(* IEC 61131-3 sources: FANUC_dev/LDJ/Kvara/PLC, 2 files *)

(* ---- Canfb.plc ---- *)
* Blocchi gestione periferiche CANopen da PLC

VAR_IN_OUT
AS_DATA0 AT %CanFb48; * CanFb48 buffer I/O Canopen
AS_DATA1 AT %CanFb49; * CanFb49 buffer I/O Canopen
AS_DATA2 AT %CanFb50; * CanFb50 buffer I/O Canopen
AS_DATA3 AT %CanFb51; * CanFb51 buffer I/O Canopen
AS_DATA4 AT %CanFb52; * CanFb52 buffer I/O Canopen
AS_DATA5 AT %CanFb53; * CanFb53 buffer I/O Canopen
AS_DATA6 AT %CanFb54; * CanFb54 buffer I/O Canopen
AS_DATA7 AT %CanFb55; * CanFb55 buffer I/O Canopen
DI_DATA0 AT %CanFb56; * CanFb56 Dato 0 input
DI_DATA1 AT %CanFb57; * CanFb57 Dato 1 input
DI_COBID AT %CanFb58; * CanFb58 Identificatore oggetto CanOpen
CONTROLREG AT %CanFb59; * CanFb59 registro comando (bit 0-7=codice comando)
CMD_RESET AT %CanFb59.30; * CanFb59.30 Reset nodo
CMD_ENAB AT %CanFb59.31; * CanFb59.31 Enable esecuzione comando
STATUSREG AT %CanFb60; * CanFb60 registro stato
DO_CONFIRM AT %CanFb60.31; * CanFb60.31 conferma comando eseguito
DO_ERROR AT %CanFb61; * CanFb61 codice errore comando
DO_DATA0 AT %CanFb62; * CanFb62 Dato 0 output
DO_DATA1 AT %CanFb63; * CanFb63 Dato 1 output
END_VAR

* -------------------------------------------------------*
* Blocco Funzionale generico invio comando a nodo CANopen
* -------------------------------------------------------*

FUNCTION_BLOCK COP_COMMAND

VAR_INPUT
CM_ENAB: BOOL; * Richiesta esecuzione comando
CM_RESET: BOOL; * Richiesta di reset del nodo
CM_CODE: DWORD; * Codice del comando
CI_COBID: DWORD; * Identificatore oggetto CanOpen
CI_DATA0: DWORD; * Dato 0 in input
CI_DATA1: DWORD; * Dato 1 in input
END_VAR

VAR_OUTPUT
CS_CONFIRM: BOOL; * Conferma comando eseguito
CO_ERROR: WORD; * Codice di errore
CO_ERRORINFO: DWORD; * Informazioni aggiuntive su errore
CO_DATA0: DWORD; * Dato 0 in output
CO_DATA1: DWORD; * Dato 1 in output
CO_DATA2: DWORD; * Dato 2 in output
CO_DATA3: DWORD; * Dato 3 in output
CO_DATA4: DWORD; * Dato 4 in output
CO_DATA5: DWORD; * Dato 5 in output
CO_DATA6: DWORD; * Dato 6 in output
CO_DATA7: DWORD; * Dato 7 in output
CO_DATA8: DWORD; * Dato 8 in output
END_VAR

VAR
StPrecEnab: BOOL; * Stato precedente ingresso ENAB
StPrecReset: BOOL; * Stato precedente ingresso RESET
StPrecConfirm: BOOL; * Stato precedente segnale CONFIRM
RTEnab: BOOL; * Fronte salita ingresso ENAB
MemCmdInProg: BOOL; * Mem. comando in corso
MemErrBusy: BOOL; * Mem. errore area comandi occupata
CmdFinished: BOOL; * Conferma comando terminato
END_VAR

* Sul fronte di salita del comando, copia tutti i dati in andata

LD   CM_ENAB      ** Richiesta esecuzione comando
ANDN StPrecEnab   ** Stato precedente ingresso ENAB
ST   RTEnab       ** Fronte salita ingresso ENAB

LD   RTEnab       ** Fronte salita ingresso ENAB
ANDN CMD_ENAB     ** CanFb59.31 Enable esecuzione comando
ANDN DO_CONFIRM   ** CanFb60.31 conferma comando eseguito
S    MemCmdInProg ** Mem. comando in corso

LDN  CM_ENAB      ** Richiesta esecuzione comando
ANDN CMD_ENAB     ** CanFb59.31 Enable esecuzione comando
ANDN DO_CONFIRM   ** CanFb60.31 conferma comando eseguito
OR   CM_RESET     ** Richiesta di reset del nodo
R    MemCmdInProg ** Mem. comando in corso

LD   RTEnab       ** Fronte salita ingresso ENAB
ANDN MemCmdInProg ** Mem. comando in corso
S    MemErrBusy   ** Mem. errore area comandi occupata

LDN  CM_ENAB      ** Richiesta esecuzione comando
R    MemErrBusy   ** Mem. errore area comandi occupata

LD   RTEnab       ** Fronte salita ingresso ENAB
AND  MemCmdInProg ** Mem. comando in corso
JMPCN END_COMMAND

LD   CONTROLREG   ** CanFb59 registro comando (bit 0-7=codice comando)
AND  16#FFFFFF00
OR   CM_CODE      ** Codice del comando
ST   CONTROLREG   ** CanFb59 registro comando (bit 0-7=codice comando)

LD   CI_COBID     ** Identificatore oggetto CanOpen
ST   DI_COBID     ** CanFb58 Identificatore oggetto CanOpen

LD   CM_CODE      ** Codice del comando
EQ   4            * PDO SEND
JMPC PDO_SEND_CMD

LD   CI_DATA0     ** Dato 0 in input
ST   DI_DATA0     ** CanFb56 Dato 0 input

LD   CI_DATA1     ** Dato 1 in input
ST   DI_DATA1     ** CanFb57 Dato 1 input

JMP  END_COMMAND

PDO_SEND_CMD:
LD   DI_COBID     ** CanFb58 Identificatore oggetto CanOpen
AND  16#FFFF00FF  * Mask offset
OR   16#3000      * Offset AS_DATA0 (48)
ST   DI_COBID     ** CanFb58 Identificatore oggetto CanOpen

LD   CI_DATA0     ** Dato 0 in input
ST   AS_DATA0     ** CanFb48 buffer I/O Canopen

LD   CI_DATA1     ** Dato 1 in input
ST   AS_DATA1     ** CanFb49 buffer I/O Canopen

END_COMMAND:

LD   CM_ENAB      ** Richiesta esecuzione comando
ST   StPrecEnab   ** Stato precedente ingresso ENAB

* Scrive i bit di ENAB e RESET

LD   MemCmdInProg ** Mem. comando in corso
JMPCN END_CMD_ENAB

LD   CM_ENAB      ** Richiesta esecuzione comando
ST   CMD_ENAB     ** CanFb59.31 Enable esecuzione comando

END_CMD_ENAB:

LD   CM_RESET     ** Richiesta di reset del nodo
OR   StPrecReset  ** Stato precedente ingresso RESET
JMPCN END_RESET

LD   CM_RESET     ** Richiesta di reset del nodo
ST   CMD_RESET    ** CanFb59.30 Reset nodo

LD   %PLCFLAGS.0
ST   CMD_ENAB     ** CanFb59.31 Enable esecuzione comando

END_RESET:

LD   CM_RESET     ** Richiesta di reset del nodo
ST   StPrecReset  ** Stato precedente ingresso RESET

* Sul fronte di salita della conferma fine comando, legge tutti i dati di ritorno

LD   DO_CONFIRM   ** CanFb60.31 conferma comando eseguito
AND  MemCmdInProg ** Mem. comando in corso
ST   CmdFinished  ** Conferma comando terminato

LD   DO_CONFIRM   ** CanFb60.31 conferma comando eseguito
ANDN StPrecConfirm ** Stato precedente segnale CONFIRM
AND  CmdFinished  ** Conferma comando terminato
JMPCN END_DATA

LD   DO_ERROR     ** CanFb61 codice errore comando
ST   CO_ERROR     ** Codice di errore

LD   DO_ERROR     ** CanFb61 codice errore comando
NE   0
JMPC TAKE_ERRINFO

LD   0
ST   CO_ERRORINFO ** Informazioni aggiuntive su errore

LD   CM_CODE      ** Codice del comando
EQ   5            * PDO READ
OR   (
LD   CM_CODE      ** Codice del comando
EQ   9            * SDO READSTR
)
OR   (
LD   CM_CODE      ** Codice del comando
EQ   10           * HISTORY ALARM
)
JMPC PDO_READ_CMD

LD   DO_DATA0     ** CanFb62 Dato 0 output
ST   CO_DATA0     ** Dato 0 in output

LD   DO_DATA1     ** CanFb63 Dato 1 output
ST   CO_DATA1     ** Dato 1 in output

JMP  END_DATA

PDO_READ_CMD:

LD   DO_DATA0     ** CanFb62 Dato 0 output
ST   CO_DATA0     ** Dato 0 in output

LD   AS_DATA0     ** CanFb48 buffer I/O Canopen
ST   CO_DATA1     ** Dato 1 in output

LD   AS_DATA1     ** CanFb49 buffer I/O Canopen
ST   CO_DATA2     ** Dato 2 in output

LD   CM_CODE      ** Codice del comando
EQ   5            * PDO READ
JMPC END_DATA

LD   AS_DATA2     ** CanFb50 buffer I/O Canopen
ST   CO_DATA3     ** Dato 3 in output

LD   AS_DATA3     ** CanFb51 buffer I/O Canopen
ST   CO_DATA4     ** Dato 4 in output

LD   AS_DATA4     ** CanFb52 buffer I/O Canopen
ST   CO_DATA5     ** Dato 5 in output

LD   AS_DATA5     ** CanFb53 buffer I/O Canopen
ST   CO_DATA6     ** Dato 6 in output

LD   AS_DATA6     ** CanFb54 buffer I/O Canopen
ST   CO_DATA7     ** Dato 7 in output

LD   AS_DATA7     ** CanFb55 buffer I/O Canopen
ST   CO_DATA8     ** Dato 8 in output

JMP  END_DATA

TAKE_ERRINFO:

LD   DO_DATA0     ** CanFb62 Dato 0 output
ST   CO_ERRORINFO ** Informazioni aggiuntive su errore

LD   0
ST   CO_DATA0     ** Dato 0 in output
ST   CO_DATA1     ** Dato 1 in output

END_DATA:

LD   MemErrBusy   ** Mem. errore area comandi occupata
JMPCN END_TR_ERR

LD   16#25        * Errore TRANSFER_BUSY
ST   CO_ERROR     ** Codice di errore

END_TR_ERR:

* Scrive in output la conferma

LD   DO_CONFIRM   ** CanFb60.31 conferma comando eseguito
ST   StPrecConfirm ** Stato precedente segnale CONFIRM

LD   CmdFinished  ** Conferma comando terminato
OR   MemErrBusy   ** Mem. errore area comandi occupata
ST   CS_CONFIRM   ** Conferma comando eseguito

END_FUNCTION_BLOCK

* -------------------------------------------------------*
* Comando di cambio di stato a nodo CANopen
* -------------------------------------------------------*

FUNCTION_BLOCK COP_NMT

VAR_INPUT
CM_ENAB: BOOL; * Richiesta esecuzione comando
CM_RESET: BOOL; * Richiesta di reset del nodo
CI_STATE: DWORD; * Stato richiesto
END_VAR

VAR_OUTPUT
CS_CONFIRM: BOOL; * Conferma comando eseguito
CO_ERROR: WORD; * Codice di errore
END_VAR

VAR
COPFB: COP_COMMAND;
END_VAR

LD   CM_ENAB      ** Richiesta esecuzione comando
ST   COPFB.CM_ENAB

LD   CM_RESET     ** Richiesta di reset del nodo
ST   COPFB.CM_RESET

LD   1
ST   COPFB.CM_CODE

LD   CI_STATE     ** Stato richiesto
ST   COPFB.CI_DATA0

CAL  COPFB

LD   COPFB.CS_CONFIRM
ST   CS_CONFIRM   ** Conferma comando eseguito

LD   COPFB.CO_ERROR
ST   CO_ERROR     ** Codice di errore

END_FUNCTION_BLOCK

* -------------------------------------------------------*
* Comando di lettura SDO a nodo CANopen
* -------------------------------------------------------*

FUNCTION_BLOCK COP_SDO_READ

VAR_INPUT
CM_ENAB: BOOL; * Richiesta esecuzione comando
CM_RESET: BOOL; * Richiesta di reset del nodo
CI_INDEX: DWORD; * Numero index dato da leggere
CI_SUBINDEX: DWORD; * Numero subindex dato da leggere
END_VAR

VAR_OUTPUT
CS_CONFIRM: BOOL; * Conferma comando eseguito
CO_ERROR: WORD; * Codice di errore
CO_ERRORINFO: DWORD; * Informazioni aggiuntive su errore
CO_DATALENGTH: DWORD; * Lunghezza dato letto in byte
CO_DATA0: DWORD; * Valore del dato letto
END_VAR

VAR
COPFB: COP_COMMAND;
END_VAR

LD   CM_ENAB      ** Richiesta esecuzione comando
ST   COPFB.CM_ENAB

LD   CM_RESET     ** Richiesta di reset del nodo
ST   COPFB.CM_RESET

LD   2
ST   COPFB.CM_CODE

LD   CI_INDEX     ** Numero index dato da leggere
SHL  16
OR   (
LD   CI_SUBINDEX  ** Numero subindex dato da leggere
SHL  8
)
ST   COPFB.CI_COBID

CAL  COPFB

LD   COPFB.CS_CONFIRM
ST   CS_CONFIRM   ** Conferma comando eseguito

LD   COPFB.CO_ERROR
ST   CO_ERROR     ** Codice di errore

LD   COPFB.CO_ERRORINFO
ST   CO_ERRORINFO ** Informazioni aggiuntive su errore

LD   COPFB.CO_DATA0
ST   CO_DATALENGTH ** Lunghezza dato letto in byte

LD   COPFB.CO_DATA1
ST   CO_DATA0     ** Valore del dato letto

END_FUNCTION_BLOCK

* -------------------------------------------------------*
* Comando di scrittura SDO a nodo CANopen
* -------------------------------------------------------*

FUNCTION_BLOCK COP_SDO_WRITE

VAR_INPUT
CM_ENAB: BOOL; * Richiesta esecuzione comando
CM_RESET: BOOL; * Richiesta di reset del nodo
CI_INDEX: DWORD; * Numero index dato da scrivere
CI_SUBINDEX: DWORD; * Numero subindex dato da scrivere
CI_DATALENGTH: DWORD; * Lunghezza dato da scrivere in byte
CI_DATA0: DWORD; * Valore da scrivere
END_VAR

VAR_OUTPUT
CS_CONFIRM: BOOL; * Conferma comando eseguito
CO_ERROR: WORD; * Codice di errore
CO_ERRORINFO: DWORD; * Informazioni aggiuntive su errore
END_VAR

VAR
COPFB: COP_COMMAND;
END_VAR

LD   CM_ENAB      ** Richiesta esecuzione comando
ST   COPFB.CM_ENAB

LD   CM_RESET     ** Richiesta di reset del nodo
ST   COPFB.CM_RESET

LD   3
ST   COPFB.CM_CODE

LD   CI_INDEX     ** Numero index dato da scrivere
SHL  16
OR   (
LD   CI_SUBINDEX  ** Numero subindex dato da scrivere
SHL  8
)
OR   CI_DATALENGTH ** Lunghezza dato da scrivere in byte
ST   COPFB.CI_COBID

LD   CI_DATA0     ** Valore da scrivere
ST   COPFB.CI_DATA0

CAL  COPFB

LD   COPFB.CS_CONFIRM
ST   CS_CONFIRM   ** Conferma comando eseguito

LD   COPFB.CO_ERROR
ST   CO_ERROR     ** Codice di errore

LD   COPFB.CO_ERRORINFO
ST   CO_ERRORINFO ** Informazioni aggiuntive su errore

END_FUNCTION_BLOCK

* -------------------------------------------------------*
* Comando di invio PDO a nodo CANopen
* -------------------------------------------------------*

FUNCTION_BLOCK COP_PDO_SEND

VAR_INPUT
CM_ENAB: BOOL; * Richiesta esecuzione comando
CM_RESET: BOOL; * Richiesta di reset del nodo
CI_COBID: DWORD; * Identificatore oggetto CanOpen
CI_DATALENGTH: DWORD; * Lunghezza dato da scrivere in byte
CI_DATA0: DWORD; * Valore da inviare (BYTE 0-3)
CI_DATA1: DWORD; * Valore da inviare (BYTE 4-7)
END_VAR

VAR_OUTPUT
CS_CONFIRM: BOOL; * Conferma comando eseguito
CO_ERROR: WORD; * Codice di errore
END_VAR

VAR
COPFB: COP_COMMAND;
END_VAR

LD   CM_ENAB      ** Richiesta esecuzione comando
ST   COPFB.CM_ENAB

LD   CM_RESET     ** Richiesta di reset del nodo
ST   COPFB.CM_RESET

LD   4
ST   COPFB.CM_CODE

LD   CI_COBID     ** Identificatore oggetto CanOpen
SHL  16
OR   CI_DATALENGTH ** Lunghezza dato da scrivere in byte
ST   COPFB.CI_COBID

LD   CI_DATA0     ** Valore da inviare (BYTE 0-3)
ST   COPFB.CI_DATA0

LD   CI_DATA1     ** Valore da inviare (BYTE 4-7)
ST   COPFB.CI_DATA1

CAL  COPFB

LD   COPFB.CS_CONFIRM
ST   CS_CONFIRM   ** Conferma comando eseguito

LD   COPFB.CO_ERROR
ST   CO_ERROR     ** Codice di errore

END_FUNCTION_BLOCK

* -------------------------------------------------------*
* Comando di lettura PDO da nodo CANopen
* -------------------------------------------------------*

FUNCTION_BLOCK COP_PDO_READ

VAR_INPUT
CM_ENAB: BOOL; * Richiesta esecuzione comando
CM_RESET: BOOL; * Richiesta di reset del nodo
CI_COBID: DWORD; * Identificatore oggetto CanOpen
END_VAR

VAR_OUTPUT
CS_CONFIRM: BOOL; * Conferma comando eseguito
CO_ERROR: WORD; * Codice di errore
CO_DATALENGTH: DWORD; * Lunghezza PDO letto in byte
CO_DATA0: DWORD; * Valore del dato letto (BYTE 0-3)
CO_DATA1: DWORD; * Valore del dato letto (BYTE 4-7)
END_VAR

VAR
COPFB: COP_COMMAND;
END_VAR

LD   CM_ENAB      ** Richiesta esecuzione comando
ST   COPFB.CM_ENAB

LD   CM_RESET     ** Richiesta di reset del nodo
ST   COPFB.CM_RESET

LD   5
ST   COPFB.CM_CODE

LD   CI_COBID     ** Identificatore oggetto CanOpen
SHL  16
ST   COPFB.CI_COBID

CAL  COPFB

LD   COPFB.CS_CONFIRM
ST   CS_CONFIRM   ** Conferma comando eseguito

LD   COPFB.CO_ERROR
ST   CO_ERROR     ** Codice di errore

LD   COPFB.CO_DATA0
ST   CO_DATALENGTH ** Lunghezza PDO letto in byte

LD   COPFB.CO_DATA1
ST   CO_DATA0     ** Valore del dato letto (BYTE 0-3)

LD   COPFB.CO_DATA2
ST   CO_DATA1     ** Valore del dato letto (BYTE 4-7)

END_FUNCTION_BLOCK

* -------------------------------------------------------*
* Comando di registrazione PDO
* -------------------------------------------------------*

FUNCTION_BLOCK COP_PDO_REGISTER

VAR_INPUT
CM_ENAB: BOOL; * Richiesta esecuzione comando
CM_RESET: BOOL; * Richiesta di reset del nodo
CI_COBID: DWORD; * Identificatore oggetto CanOpen
CI_DATALENGTH: DWORD; * Lunghezza in BYTE e tipo dato (FFFF = cancella registr.)
                      * lungh + 0: legge con COP_PDO_READ
                      * lungh + 256: legge da CanFb0-CanFb47
                      * lungh + 512: legge da IW0-IW2047
CI_DATAOFFSET: DWORD; * Offset rinfresco (CanFb[0-47] / IO[0-2047])
END_VAR

VAR_OUTPUT
CS_CONFIRM: BOOL; * Conferma comando eseguito
CO_ERROR: WORD; * Codice di errore
END_VAR

VAR
COPFB: COP_COMMAND;
END_VAR

LD   CM_ENAB      ** Richiesta esecuzione comando
ST   COPFB.CM_ENAB

LD   CM_RESET     ** Richiesta di reset del nodo
ST   COPFB.CM_RESET

LD   6
ST   COPFB.CM_CODE

LD   CI_COBID     ** Identificatore oggetto CanOpen
SHL  16
OR   CI_DATALENGTH ** Lunghezza in BYTE e tipo dato (FFFF = cancella registr.)
ST   COPFB.CI_COBID

LD   CI_DATAOFFSET ** Offset rinfresco (CanFb[0-47] / IO[0-2047])
ST   COPFB.CI_DATA0

CAL  COPFB

LD   COPFB.CS_CONFIRM
ST   CS_CONFIRM   ** Conferma comando eseguito

LD   COPFB.CO_ERROR
ST   CO_ERROR     ** Codice di errore

END_FUNCTION_BLOCK

* -------------------------------------------------------*
* Comando di impostazione sincronizzazione ciclica
* -------------------------------------------------------*

FUNCTION_BLOCK COP_CYCLIC_SYNC

VAR_INPUT
CM_ENAB: BOOL; * Richiesta esecuzione comando
CM_RESET: BOOL; * Richiesta di reset del nodo
CI_SYNC_TIME: DWORD; * Tempo ciclo (0=Disab, 1=Singolo, 10-250=Ciclico in ms)
END_VAR

VAR_OUTPUT
CS_CONFIRM: BOOL; * Conferma comando eseguito
CO_ERROR: WORD; * Codice di errore
END_VAR

VAR
COPFB: COP_COMMAND;
END_VAR

LD   CM_ENAB      ** Richiesta esecuzione comando
ST   COPFB.CM_ENAB

LD   CM_RESET     ** Richiesta di reset del nodo
ST   COPFB.CM_RESET

LD   7
ST   COPFB.CM_CODE

LD   CI_SYNC_TIME ** Tempo ciclo (0=Disab, 1=Singolo, 10-250=Ciclico in ms)
ST   COPFB.CI_DATA0

CAL  COPFB

LD   COPFB.CS_CONFIRM
ST   CS_CONFIRM   ** Conferma comando eseguito

LD   COPFB.CO_ERROR
ST   CO_ERROR     ** Codice di errore

END_FUNCTION_BLOCK

* -------------------------------------------------------*
* Comando di remote request oggetto CANopen
* -------------------------------------------------------*

FUNCTION_BLOCK COP_REM_REQUEST

VAR_INPUT
CM_ENAB: BOOL; * Richiesta esecuzione comando
CM_RESET: BOOL; * Richiesta di reset del nodo
CI_COBID: DWORD; * Identificatore oggetto CanOpen
END_VAR

VAR_OUTPUT
CS_CONFIRM: BOOL; * Conferma comando eseguito
CO_ERROR: WORD; * Codice di errore
END_VAR

VAR
COPFB: COP_COMMAND;
END_VAR

LD   CM_ENAB      ** Richiesta esecuzione comando
ST   COPFB.CM_ENAB

LD   CM_RESET     ** Richiesta di reset del nodo
ST   COPFB.CM_RESET

LD   8
ST   COPFB.CM_CODE

LD   CI_COBID     ** Identificatore oggetto CanOpen
ST   COPFB.CI_COBID

CAL  COPFB

LD   COPFB.CS_CONFIRM
ST   CS_CONFIRM   ** Conferma comando eseguito

LD   COPFB.CO_ERROR
ST   CO_ERROR     ** Codice di errore

END_FUNCTION_BLOCK

* -------------------------------------------------------*
* Comando di lettura SDO su stringa da nodo CANopen
* -------------------------------------------------------*

FUNCTION_BLOCK COP_SDO_READSTRING

VAR_INPUT
CM_ENAB: BOOL; * Richiesta esecuzione comando
CM_RESET: BOOL; * Richiesta di reset del nodo
CI_INDEX: DWORD; * Numero index dato da leggere
CI_SUBINDEX: DWORD; * Numero subindex dato da leggere
END_VAR

VAR_OUTPUT
CS_CONFIRM: BOOL; * Conferma comando eseguito
CO_ERROR: WORD; * Codice di errore
CO_ERRORINFO: DWORD; * Informazioni aggiuntive su errore
CO_DATALENGTH: DWORD; * Lunghezza stringa letta in byte
CO_DATA0: DWORD; * Stringa letta (BYTE 0-3)
CO_DATA1: DWORD; * Stringa letta (BYTE 4-7)
CO_DATA2: DWORD; * Stringa letta (BYTE 8-11)
CO_DATA3: DWORD; * Stringa letta (BYTE 12-15)
CO_DATA4: DWORD; * Stringa letta (BYTE 16-19)
CO_DATA5: DWORD; * Stringa letta (BYTE 20-23)
CO_DATA6: DWORD; * Stringa letta (BYTE 24-27)
CO_DATA7: DWORD; * Stringa letta (BYTE 28-31)
END_VAR

VAR
COPFB: COP_COMMAND;
END_VAR

LD   CM_ENAB      ** Richiesta esecuzione comando
ST   COPFB.CM_ENAB

LD   CM_RESET     ** Richiesta di reset del nodo
ST   COPFB.CM_RESET

LD   9
ST   COPFB.CM_CODE

LD   CI_INDEX     ** Numero index dato da leggere
SHL  16
OR   (
LD   CI_SUBINDEX  ** Numero subindex dato da leggere
SHL  8
)
ST   COPFB.CI_COBID

CAL  COPFB

LD   COPFB.CS_CONFIRM
ST   CS_CONFIRM   ** Conferma comando eseguito

LD   COPFB.CO_ERROR
ST   CO_ERROR     ** Codice di errore

LD   COPFB.CO_ERRORINFO
ST   CO_ERRORINFO ** Informazioni aggiuntive su errore

LD   COPFB.CO_DATA0
ST   CO_DATALENGTH ** Lunghezza stringa letta in byte

LD   COPFB.CO_DATA1
ST   CO_DATA0     ** Stringa letta (BYTE 0-3)

LD   COPFB.CO_DATA2
ST   CO_DATA1     ** Stringa letta (BYTE 4-7)

LD   COPFB.CO_DATA3
ST   CO_DATA2     ** Stringa letta (BYTE 8-11)

LD   COPFB.CO_DATA4
ST   CO_DATA3     ** Stringa letta (BYTE 12-15)

LD   COPFB.CO_DATA5
ST   CO_DATA4     ** Stringa letta (BYTE 16-19)

LD   COPFB.CO_DATA6
ST   CO_DATA5     ** Stringa letta (BYTE 20-23)

LD   COPFB.CO_DATA7
ST   CO_DATA6     ** Stringa letta (BYTE 24-27)

LD   COPFB.CO_DATA8
ST   CO_DATA7     ** Stringa letta (BYTE 28-31)

END_FUNCTION_BLOCK

* -------------------------------------------------------*
* Comando Read/Reset History alarm da nodo CANopen
* -------------------------------------------------------*

FUNCTION_BLOCK COP_ALARMS_HIST

VAR_INPUT
CM_ENAB:  BOOL; * Richiesta esecuzione comando
CM_RESET: BOOL; * Richiesta di reset del nodo
CI_MODE:  BOOL; * 0=Read  1=Read & Reset
END_VAR

VAR_OUTPUT
CS_CONFIRM: BOOL; * Conferma comando eseguito
CO_ERROR:   WORD; * Codice di errore
CO_ERRORINFO: DWORD;  * Informazioni aggiuntive su errore
CO_ALARMS:    DWORD;  * Numero di allarmi presenti
CO_ALRM1: DWORD; * Ultimo allarme "n"
CO_ALRM2: DWORD; * Allarme "n-1"
CO_ALRM3: DWORD; * Allarme "n-2"
CO_ALRM4: DWORD; * Allarme "n-3"
CO_ALRM5: DWORD; * Allarme "n-4"
CO_ALRM6: DWORD; * Allarme "n-5"
CO_ALRM7: DWORD; * Allarme "n-6"
CO_ALRM8: DWORD; * Allarme "n-7"
END_VAR

VAR
COPFB: COP_COMMAND;
END_VAR

LD   CM_ENAB      ** Richiesta esecuzione comando
ST   COPFB.CM_ENAB

LD   CM_RESET     ** Richiesta di reset del nodo
ST   COPFB.CM_RESET

LD   10
ST   COPFB.CM_CODE

LD   CI_MODE      ** 0=Read  1=Read & Reset
ST   COPFB.CI_DATA0.0   ** CanFb56 Dato 0 input

CAL  COPFB

LD   COPFB.CS_CONFIRM
ST   CS_CONFIRM   ** Conferma comando eseguito

LD   COPFB.CO_ERROR
ST   CO_ERROR     ** Codice di errore

LD   COPFB.CO_ERRORINFO
ST   CO_ERRORINFO ** Informazioni aggiuntive su errore

LD   DO_DATA0     ** CanFb62 Dato 0 output
ST   CO_ALARMS    ** Numero di allarmi presenti

LD   COPFB.CO_DATA1
ST   CO_ALRM1     ** Ultimo allarme "n"

LD   COPFB.CO_DATA2
ST   CO_ALRM2     ** Allarme "n-1"

LD   COPFB.CO_DATA3
ST   CO_ALRM3     ** Allarme "n-2"

LD   COPFB.CO_DATA4
ST   CO_ALRM4     ** Allarme "n-3"

LD   COPFB.CO_DATA5
ST   CO_ALRM5     ** Allarme "n-4"

LD   COPFB.CO_DATA6
ST   CO_ALRM6     ** Allarme "n-5"

LD   COPFB.CO_DATA7
ST   CO_ALRM7     ** Allarme "n-6"

LD   COPFB.CO_DATA8
ST   CO_ALRM8     ** Allarme "n-7"

END_FUNCTION_BLOCK

* -------------------------------------------------------*
* Comando di lettura VACON ReadAnyParam
* -------------------------------------------------------*

FUNCTION_BLOCK VAC_PAR_READ

VAR_INPUT
CM_ENAB: BOOL; * Richiesta esecuzione comando
CM_RESET: BOOL; * Richiesta di reset del nodo
CI_INDEX: DWORD; * Numero parametro da leggere
END_VAR

VAR_OUTPUT
CS_CONFIRM: BOOL; * Conferma comando eseguito
CO_ERROR: WORD; * Codice di errore
CO_ERRORINFO: DWORD; * Informazioni aggiuntive su errore
CO_DATALENGTH: DWORD; * Lunghezza dato letto in byte
CO_DATA0: DWORD; * Valore del dato letto
END_VAR

VAR
COPFB: COP_COMMAND;
END_VAR

LD   CM_ENAB      ** Richiesta esecuzione comando
ST   COPFB.CM_ENAB

LD   CM_RESET     ** Richiesta di reset del nodo
ST   COPFB.CM_RESET

LD   255
ST   COPFB.CM_CODE

LD   CI_INDEX     ** Numero index dato da leggere
ST   COPFB.CI_COBID

CAL  COPFB

LD   COPFB.CS_CONFIRM
ST   CS_CONFIRM   ** Conferma comando eseguito

LD   COPFB.CO_ERROR
ST   CO_ERROR     ** Codice di errore

LD   COPFB.CO_ERRORINFO
ST   CO_ERRORINFO ** Informazioni aggiuntive su errore

LD   COPFB.CO_DATA0
ST   CO_DATALENGTH ** Lunghezza dato letto in byte

LD   COPFB.CO_DATA1
ST   CO_DATA0     ** Valore del dato letto

END_FUNCTION_BLOCK

* -------------------------------------------------------*
* Comando di scrittura VACON WriteAnyParam
* -------------------------------------------------------*

FUNCTION_BLOCK VAC_PAR_WRITE

VAR_INPUT
CM_ENAB: BOOL; * Richiesta esecuzione comando
CM_RESET: BOOL; * Richiesta di reset del nodo
CI_INDEX: DWORD; * Numero parametro dato da scrivere
CI_DATA0: DWORD; * Valore da scrivere
END_VAR

VAR_OUTPUT
CS_CONFIRM: BOOL; * Conferma comando eseguito
CO_ERROR: WORD; * Codice di errore
CO_ERRORINFO: DWORD; * Informazioni aggiuntive su errore
END_VAR

VAR
COPFB: COP_COMMAND;
END_VAR

LD   CM_ENAB      ** Richiesta esecuzione comando
ST   COPFB.CM_ENAB

LD   CM_RESET     ** Richiesta di reset del nodo
ST   COPFB.CM_RESET

LD   254
ST   COPFB.CM_CODE

LD   CI_INDEX     ** Numero index dato da scrivere
ST   COPFB.CI_COBID

LD   CI_DATA0     ** Valore da scrivere
ST   COPFB.CI_DATA0

CAL  COPFB

LD   COPFB.CS_CONFIRM
ST   CS_CONFIRM   ** Conferma comando eseguito

LD   COPFB.CO_ERROR
ST   CO_ERROR     ** Codice di errore

LD   COPFB.CO_ERRORINFO
ST   CO_ERRORINFO ** Informazioni aggiuntive su errore

END_FUNCTION_BLOCK

(* ---- usercmd.plc ---- *)
* File USERCMD.PLC

#include "iof.inc"
#include "iol.inc"
#include "mem.inc"

VAR
IN_LUBR_ERR    AT %IW0.13;  * IW0.13 Errore Centralina Lubrificazione (cartuccia Vuota)
LUBR_ERR: BOOL;              * IW0.13 Errore Centralina Lubrificazione (cartuccia Vuota) Solo quando lubrificazzione in corso
LUBR_OK     AT %IW0.14;  * IW0.14 Lubrificazione OK
IN_CELLA_APERTA AT %IW3.8; * IW3.8 Ingresso Cella Aperta
BRAKE_OPEN  AT %IW3.0;   * IW3.0 Freni aperti, consenso al movimento Ok
STOP_PCV    AT %IW3.3;   * IW3.3 Blocco ciclo al PCV
STOP_PCL    AT %IW3.4;   * IW3.4 Blocco ciclo al PCL dopo il rinculo
STOP_PMI    AT %IW3.5;   * IW3.5 Blocco ciclo al PMI dopo il tempo sosta
LUBR_REQ    AT %QW1.8;   * QW1.8 Richiesta Lubrificazione
FIRST_BEND  AT %QW2.13;  * QW2.13 Prima Piega Attiva
PMS_ROBOT   AT %QW2.8;   * QW2.8 PMS per Robot
OUT_INT_LAMP AT %QW1.10; * QW1.10 Uscita Accensione Lampada Interna
PUMP_ON_PUNCH_HOLDER AT %QW1.11; * Uscita Attivazione Pompa Bloccaggi Superiori
PUMP_ON_DIE_HOLDER   AT %QW1.12; * Uscita Attivazione Pompa Bloccaggi Inferiori o Bloccaggio Singolo
HOLDER_OPENED        AT %QW1.13; * Uscita Bloccaggi Aperti
PUNCH_HOLDER_OPENED  AT %QW1.14; * Uscita Bloccaggi Superiori Aperti
DIE_HOLDER_OPENED    AT %QW1.15; * Uscita Bloccaggi Inferiori Aperti
ANIN2       AT %IW51;    * Ingresso analogico Pin 2
ANIN3       AT %IW52;    * Ingresso analogico Pin 3
VOLT_LED    AT %QW102;   * QW102 Tensione regolazione intensità luminosa Lampada

Cond_Cont_Lubr: BOOL; * Condizione Conteggio Lubrificazione
Cond_Reload_Cont: BOOL; * Condizione Reload Conteggio Lubrificazione
Param_Changed: BOOL; * Parametro Cambiato
LUB_ERR_REMIND: BOOL; * Reminder Cartuccia Lubrificazione Terminata
LubrErr: BOOL; * Cartuccia Vuota
Lubrinproc: BOOL; * Cartuccia Vuota stato in memoria
VLED_0_BIT: WORD; * Tensione Lampada 0% in Bit
VLED_100_BIT: WORD; * Tensione Lampada 100% in Bit

***** Limitazione Sbilanciamento in Discesa Lenta *****
Y1_STOP_UNBALANCE: BOOL; * Necessario Stop Y1 per sbilanciamento eccessivo
Y2_STOP_UNBALANCE: BOOL; * Necessario Stop Y2 per sbilanciamento eccessivo
Y1_FEED_CALC: WORD; * Valore Feed Y1 Ricalcolata
Y2_FEED_CALC: WORD; * Valore Feed Y2 Ricalcolata
***** Fine Limitazione Sbilanciamento in Discesa Lenta *****

TON_FILTER: TON;
#defcom TON_FILTER.Q Filtro per pedale di discesa
#defcom CTD_LUBR.Q Fine Conteggio per attivazione lubrificazione
#defcom CTD_LUBR.CV Stato del Contatore Lubrificazione
CTD_LUBR: CTD;
#defcom CTD_LUBR_OK.Q Fine Conteggio per check lubrificazione
CTD_LUBR_OK: CTD;
#defcom TP_LUBR.Q    Tempo Uscita Lubrificazione Attiva
TP_LUBR: TP;
#defcom TOF_LUBR_EMPTY.Q    Cartuccia Vuota
TOF_LUBR_EMPTY: TOF;
#defcom R_TRIG_LUBR.Q Fronte salita Richiesta Lubrificazione
R_TRIG_LUBR: R_TRIG;
#defcom TRIG_LUBR_OK.Q Fronte salita Ingresso Lubrificazione in corso
TRIG_LUBR_OK: TRIG;
#defcom F_TRIG_LUBREMPTY.Q Fronte discesa Cartuccia vuota
F_TRIG_LUBREMPTY: F_TRIG;

#defcom TOF_PRES_SUP.Q    Filtro apertura bloccaggi superiori
TOF_PRES_SUP: TOF;
#defcom TOF_PRES_INF.Q    Filtro apertura bloccaggi inferiori
TOF_PRES_INF: TOF;

#defcom %paruser.dwuser0     Numero cicli per lubrificazione
#defcom %paruser.dwuser1     Tensione Lampada allo 0%
#defcom %paruser.dwuser2     Tensione Lampada al 100%
#defcom %paruser.buser.0     Bloccaggi Singolo
#defcom %paruser.buser.1     Bloccaggi Doppio
V_MAX_CLOSE_TOOLS AT %paruser.dwuser4;   * Tensione Massima per Attivazione Pompa
V_MIN_CLOSE_TOOLS AT %paruser.dwuser5;   * Tensione Minima per Attivazione Pompa
V_TOOLS_OPENED    AT %paruser.dwuser6;   * Tensione Utensili Aperti

#defcom %PLCerr3.3    Allarme Richiesta Lubrificazione, Centralina non risponde
#defcom %PLCerr3.4    Allarme Cartuccia Danneggiata
#defcom %PLCerr3.5    Allarme Cartuccia Vuota
#defcom %PLCerr3.6    Allarme Freni Chiusi

END_VAR

VAR_IN_OUT

INTERNAL_LIGTH  AT %R65.0;   * R65.0 Pulsante UI accensione / spegnimento Lampada interna
VOUT_LED        AT %R64;     * R64 Tensione Bit in uscita
COUNT_LUBR_MEM  AT %R63;     * R63 Parametro Conteggio Lubrificazione in Memoria
Lubrinprocmem   AT %R62.0;   * Cartuccia vuota stato in memoria
COUNT_LUBR_CV   AT %M127;    * M127 Strokes Left for Lubrification
PERC_V_LED      AT %M128;    * M128 Percentuale Tensione LED
VOLT_LED_DEC    AT %M129.0;  * M129.0 Pulsante decremento Tensione LED 1%
VOLT_LED_INC    AT %M129.1;  * M129.1 Pulsante incremento Tensione LED 1%
VOLT_LED_DEC10  AT %M129.2;  * M129.2 Pulsante decremento Tensione LED 10%
VOLT_LED_INC10  AT %M129.3;  * M129.3 Pulsante incremento Tensione LED 10%
VOLT_LED_OFF    AT %M129.4;  * M129.4 Pulsante spegnimento Lamada
VOLT_LED_100    AT %M129.5;  * M129.5 Pulsante accensione Lampada al 100%
COUNTER         AT %paruser.dwuser0; ** Numero cicli per lubrificazione

END_VAR

* Funzione utente per la gestione di input ausiliari e il forzamento
* di input per il programma MAIN.

FUNCTION USERIN

** Filtro per pedale discesa Starmatik **

*CAL   TON_FILTER(IN=%C60.0, PT=300)

*LD    TON_FILTER.Q
*ST    %C60.0

*CAL   TOF_PRES_SUP(IN=%C61.26, PT=1000)  * IN Pressostato bloccaggi superiori
*CAL   TOF_PRES_INF(IN=%C61.27, PT=1000)  * IN Pressostato bloccaggi inferiori

*LD    TOF_PRES_SUP.Q
*ST    %C61.26   * IN Pressostato bloccaggi superiori

*LD    TOF_PRES_INF.Q
*ST    %C61.27   * IN Pressostato bloccaggi inferiori

LDN    %C62.20   ** Allarme Utente 2
ST     %C62.20   ** Allarme Utente 2

END_FUNCTION

* Funzione utente per il comando di segnalazioni e uscite ausiliarie.

FUNCTION USERCMD

* Esempio
*LD   %IW0.0
*ST   %PLCerr3.0

************************** Gestione Lubrificazione ***********************************

LD   IN_LUBR_ERR     * IW0.13 Errore Centralina Lubrificazione (cartuccia Vuota)
ORN  LUBR_REQ        ** QW1.8 Richiesta Lubrificazione
ST   LUBR_ERR        * IW0.13 Errore Centralina Lubrificazione (cartuccia Vuota) Solo quando lubrificazzione in corso

LD   %paruser.dwuser0 ** Numero cicli per lubrificazione
EQ   0
JMPC NOLUBR

LD   %C70.16      ** OUT Macchina al PMS
ST   Cond_Cont_Lubr ** Condizione Conteggio Lubrificazione

LD   COUNTER      ** Parametro Conteggio Lubrificazione
EQ   COUNT_LUBR_MEM ** R63 Parametro Conteggio Lubrificazione in Memoria
JMPC PARAM_NOT_CHANGED

LD   %PLCFLAGS.1  ** Sempre a uno
ST   Param_Changed ** Parametro Cambiato

LD   COUNTER      ** Parametro Conteggio Lubrificazione
ST   COUNT_LUBR_MEM ** R63 Parametro Conteggio Lubrificazione in Memoria

PARAM_NOT_CHANGED:

LD   CTD_LUBR.Q   ** Fine Conteggio per attivazione lubrificazione
OR   Param_Changed ** Parametro Cambiato
ST   Cond_Reload_Cont ** Condizione Reload Conteggio Lubrificazione

LD   %PLCFLAGS.0  ** Sempre a zero
ST   Param_Changed ** Parametro Cambiato

CAL  CTD_LUBR(CD:=Cond_Cont_Lubr, LD:=Cond_Reload_Cont , PV:=%paruser.dwuser0) ** Condizione Conteggio Lubrificazione

CAL  TP_LUBR(IN=CTD_LUBR.Q,PT=10000) ** Fine Conteggio per attivazione lubrificazione

CAL  R_TRIG_LUBR(CLK=TP_LUBR.Q) ** Tempo Uscita Lubrificazione Attiva

CAL  F_TRIG_LUBREMPTY(CLK=LUBR_ERR) ** IW0.13 Errore Centralina Lubrificazione (cartuccia Vuota)

CAL  TRIG_LUBR_OK(CLK=LUBR_OK) ** IW0.14 Lubrificazione OK

CAL  CTD_LUBR_OK(CD:=TRIG_LUBR_OK.Q, LD:=R_TRIG_LUBR.Q , PV:=1) ** Fronte salita Ingresso Lubrificazione in corso

LD   R_TRIG_LUBR.Q ** Fronte salita Richiesta Lubrificazione
S    Lubrinprocmem ** Cartuccia vuota stato in memoria

LD   R_TRIG_LUBR.Q ** Fronte salita Richiesta Lubrificazione
OR   (
LD   Lubrinprocmem ** Cartuccia vuota stato in memoria
AND  %PLCFLAGS.8  ** Bit a uno alla prima scansione
)
S    Lubrinproc   ** Cartuccia Vuota stato in memoria

LD   CTD_LUBR_OK.Q ** Fine Conteggio per check lubrificazione
R    Lubrinprocmem ** Cartuccia vuota stato in memoria

LD   CTD_LUBR_OK.Q ** Fine Conteggio per check lubrificazione
OR   %M5.5         ** Comando stop
R    Lubrinproc   ** Cartuccia Vuota stato in memoria

LD   CTD_LUBR.CV  ** Stato del Contatore Lubrificazione
ST   COUNT_LUBR_CV ** M127 Strokes Left for Lubrification

LD   LUBR_ERR     ** IW0.13 Errore Centralina Lubrificazione (cartuccia Vuota)
ST   LubrErr      ** Cartuccia Vuota

CAL  TOF_LUBR_EMPTY(IN=LubrErr,PT=4000) ** Cartuccia Vuota

LD   Lubrinproc   ** Cartuccia Vuota stato in memoria
ANDN TP_LUBR.Q    ** Tempo Uscita Lubrificazione Attiva
ST   %PLCerr3.4   ** Allarme Cartuccia Danneggiata

LD   %PLCFLAGS.8  ** Bit a uno alla prima scansione
ANDN LUBR_ERR     ** IW0.13 Errore Centralina Lubrificazione (cartuccia Vuota)
OR   F_TRIG_LUBREMPTY.Q ** Fronte discesa Cartuccia vuota
S    LUB_ERR_REMIND ** Reminder Cartuccia Lubrificazione Terminata

LD   %M5.5        ** Comando stop
R    LUB_ERR_REMIND ** Reminder Cartuccia Lubrificazione Terminata

LD   LUB_ERR_REMIND ** Reminder Cartuccia Lubrificazione Terminata
ST   %PLCerr3.5   ** Allarme Cartuccia Vuota

LD   TP_LUBR.Q    ** Tempo Uscita Lubrificazione Attiva
ST   LUBR_REQ     ** QW1.8 Richiesta Lubrificazione

NOLUBR:

****************** Gestione Luminosità Lampada *********************

LD   %paruser.dwuser1 ** Tensione Lampada allo 0%
DIV  10
MUL  4095
DIV  1000
ST   VLED_0_BIT   ** Tensione Lampada 0% in Bit

LD   %paruser.dwuser2 ** Tensione Lampada allo 100%
DIV  10
MUL  4095
DIV  1000
ST   VLED_100_BIT ** Tensione Lampada 100% in Bit

LD   VOLT_LED_DEC ** M129.0 Pulsante decremento Tensione LED 1%
AND  (
LD   VOUT_LED     ** R64 Tensione Bit in uscita
GT   VLED_0_BIT   ** Tensione Lampada 0% in Bit
)
JMPCN NO_LED_DEC

LD   VOUT_LED     ** R64 Tensione Bit in uscita
SUB  10
ST   VOUT_LED     ** R64 Tensione Bit in uscita

NO_LED_DEC:

LD   VOLT_LED_INC ** M129.1 Pulsante incremento Tensione LED 1%
AND  (
LD   VOUT_LED     ** R64 Tensione Bit in uscita
LT   VLED_100_BIT ** Tensione Lampada 100% in Bit
)
JMPCN NO_LED_INC

LD   VOUT_LED     ** R64 Tensione Bit in uscita
ADD  10
ST   VOUT_LED     ** R64 Tensione Bit in uscita

NO_LED_INC:

LD   VOLT_LED_DEC10 ** M129.2 Pulsante decremento Tensione LED 10%
AND  (
LD   VOUT_LED     ** R64 Tensione Bit in uscita
GT   VLED_0_BIT   ** Tensione Lampada 0% in Bit
)
JMPCN NO_LED_DEC10

LD   VOUT_LED     ** R64 Tensione Bit in uscita
SUB  50
ST   VOUT_LED     ** R64 Tensione Bit in uscita

NO_LED_DEC10:

LD   VOLT_LED_INC10 ** M129.3 Pulsante incremento Tensione LED 10%
AND  (
LD   VOUT_LED     ** R64 Tensione Bit in uscita
LT   VLED_100_BIT ** Tensione Lampada 100% in Bit
)
JMPCN NO_LED_INC10

LD   VOUT_LED     ** R64 Tensione Bit in uscita
ADD  50
ST   VOUT_LED     ** R64 Tensione Bit in uscita

NO_LED_INC10:

LD   VOLT_LED_OFF ** M129.4 Pulsante spegnimento Lamada
JMPCN LED_OFF

LD   VLED_0_BIT   ** Tensione Lampada 0% in Bit
ST   VOUT_LED     ** R64 Tensione Bit in uscita

LED_OFF:

LD   VOLT_LED_100 ** M129.5 Pulsante accensione Lampada al 100%
JMPCN LED_100

LD   VLED_100_BIT ** Tensione Lampada 100% in Bit
ST   VOUT_LED     ** R64 Tensione Bit in uscita

LED_100:

LD   VOUT_LED     ** R64 Tensione Bit in uscita
SUB  VLED_0_BIT   ** Tensione Lampada 0% in Bit
MUL  100
DIV  (
LD   VLED_100_BIT ** Tensione Lampada 100% in Bit
SUB  VLED_0_BIT   ** Tensione Lampada 0% in Bit
)
*DIV  4095
ST   PERC_V_LED   ** M128 Percentuale Tensione LED

LD   VOUT_LED     ** R64 Tensione Bit in uscita
ST   VOLT_LED     ** QW102 Tensione regolazione intensità luminosa Lampada

LD   INTERNAL_LIGTH   ** R65.0 Pulsante UI accensione / spegnimento Lampada interna
ST   OUT_INT_LAMP     ** QW1.10 Uscita Accensione Lampada Interna

******************************BLOCCO VELOCITA' IN CASO DI CELLA APERTA******************

LD      %C32.22            **LIMITAZIONE VELOCITà LAVORO
OR      IN_CELLA_APERTA    **INGRESSO CELLA APERTA
ST      %C32.22            **LIMITAZIONE VELOCITà LAVORO

******************************USCITA PIEGA CORRENTE NUMERO1*****************************

LD      %M6.27           ** Prima piega del pezzo attiva (ad uso PLC cliente)
EQ      1
ST      FIRST_BEND            **NUMERO PIEGA ATTIVA 1
****************************************************************************************
****************************** Stop Mute ************************************

LD      STOP_PCV         ** IW3.3 Blocco ciclo al PCV
ST      %M15.0           ** Blocco ciclo al PCV

LD      %C70.8           ** OUT Configurazione valvole bit 0
ANDN    (
LD      %C70.17          ** OUT Macchina al PCV
AND     %C60.0           ** IN Pedale discesa
AND     %M15.0           ** Blocco ciclo al PCV
)
ST      %C70.8           ** OUT Configurazione valvole bit 0

LD      %C70.9           ** OUT Configurazione valvole bit 1
ANDN    (
LD      %C70.17          ** OUT Macchina al PCV
AND     %C60.0           ** IN Pedale discesa
AND     %M15.0           ** Blocco ciclo al PCV
)
ST      %C70.9           ** OUT Configurazione valvole bit 1

****************************** Stop Pinch ************************************

LD      STOP_PCL         ** IW3.4 Blocco ciclo al PCL dopo il rinculo
ST      %M15.1           ** Blocco ciclo al PCL dopo il rinculo

****************************** Stop BDC ************************************

LD      STOP_PMI         ** IW3.5 Blocco ciclo al PMI dopo il tempo sosta
ST      %M15.3           ** Blocco ciclo al PMI dopo il tempo sosta

LD    %C70.16            ** OUT Macchina al PMS
ST    PMS_ROBOT          ** QW2.8 PMS per Robot

***** Limitazione Sbilanciamento in Discesa Lenta *****

LD    0            * disabilita override canale
ST    %cn0.rc2     * override pestone

LD    %ax0.ra4     * Quota attuale Y1
LT    (
LD    %ax1.ra4     * Quota attuale Y2
SUB   1000
)
AND   %M3.1        ** Discesa lavoro in corso
ST    Y1_STOP_UNBALANCE  * Necessario Stop Y1 per sbilanciamento eccessivo

LD    %ax1.ra4     * Quota attuale Y2
LT    (
LD    %ax0.ra4     * Quota attuale Y1
SUB   1000
)
AND   %M3.1        ** Discesa lavoro in corso
ST    Y2_STOP_UNBALANCE  * Necessario Stop Y2 per sbilanciamento eccessivo

LD    Y1_STOP_UNBALANCE  * Necessario Stop Y1 per sbilanciamento eccessivo
JMPC  CONTROL_UNBAL_Y1

LD    100000000
ST    %ax0.ra49           ** Feed Alta Risoluzione Y1

JMP   UNBAL_Y1_OK

CONTROL_UNBAL_Y1:

LD    %pst5              ** PAR-PLC Correzione sbilanciamento
MUL   100000
DIV   %C131              ** AX_PLC Differenza fra Y1 ed Y2
SUB   100000
ST    Y1_FEED_CALC       ** Valore Feed Y1 Ricalcolata

LD    Y1_FEED_CALC       ** Valore Feed Y1 Ricalcolata
LE    0
JMPCN FEED_Y1_ZERO

LD   0
ST   %ax0.ra49           ** Feed Alta Risoluzione Y1
ST   %ax1.ra49           ** Feed Alta Risoluzione Y2

JMP  UNBAL_Y1_OK

FEED_Y1_ZERO:

LD   Y1_FEED_CALC        ** Valore Feed Y1 Ricalcolata
ST   %ax0.ra49           ** Feed Alta Risoluzione Y1
ST   %ax1.ra49           ** Feed Alta Risoluzione Y2

UNBAL_Y1_OK:

LD    Y2_STOP_UNBALANCE  * Necessario Stop Y2 per sbilanciamento eccessivo
JMPC  CONTROL_UNBAL_Y2

LD    100000000
ST    %ax1.ra49           ** Feed Alta Risoluzione Y2

JMP   UNBAL_Y2_OK

CONTROL_UNBAL_Y2:

LD    %pst5              ** PAR-PLC Correzione sbilanciamento
MUL   100000
DIV   %C131              ** AX_PLC Differenza fra Y1 ed Y2
SUB   100000
ST    Y2_FEED_CALC       ** Valore Feed Y2 Ricalcolata

LD    Y2_FEED_CALC       ** Valore Feed Y2 Ricalcolata
LE    0
JMPCN FEED_Y2_ZERO

LD   0
ST   %ax0.ra49           ** Feed Alta Risoluzione Y1
ST   %ax1.ra49           ** Feed Alta Risoluzione Y2

JMP  UNBAL_Y2_OK

FEED_Y2_ZERO:

LD   Y2_FEED_CALC        ** Valore Feed Y2 Ricalcolata
ST   %ax0.ra49           ** Feed Alta Risoluzione Y1
ST   %ax1.ra49           ** Feed Alta Risoluzione Y2

UNBAL_Y2_OK:

***** Fine Limitazione Sbilanciamento in Discesa Lenta *****

LD    BRAKE_OPEN         ** IW3.0 Freni aperti, consenso al movimento Ok
JMPC  BRAKE_CLOSED

LD    0
ST    %ax0.ra49           ** Feed Alta Risoluzione Y1
ST    %ax1.ra49           ** Feed Alta Risoluzione Y2

BRAKE_CLOSED:

LDN   BRAKE_OPEN         ** IW3.0 Freni aperti, consenso al movimento Ok
ST    %PLCerr3.6         ** Allarme Freni Chiusi

*****Gestione Bloccaggi*****

LDN   %paruser.buser.0   ** Bloccaggi Singolo
JMPC  DOUBLE_LOCK

LD    10000000
DIV   4095
MUL   ANIN2              ** Ingresso analogico Pin 2
DIV   1000
LT    V_MIN_CLOSE_TOOLS  ** Tensione Minima per Attivazione Pompa
S     PUMP_ON_DIE_HOLDER ** Uscita Attivazione Pompa Bloccaggi Inferiori o Bloccaggio Singolo

LD    10000000
DIV   4095
MUL   ANIN2              ** Ingresso analogico Pin 2
DIV   1000
GT    V_MAX_CLOSE_TOOLS  ** Tensione Massima per Attivazione Pompa
R     PUMP_ON_DIE_HOLDER ** Uscita Attivazione Pompa Bloccaggi Inferiori o Bloccaggio Singolo

LD    10000000
DIV   4095
MUL   ANIN2              ** Ingresso analogico Pin 2
DIV   1000
GT    V_TOOLS_OPENED     ** Tensione Utensili Aperti
ST    HOLDER_OPENED      ** Uscita Bloccaggi Aperti

JMP   NO_LOCK

DOUBLE_LOCK:

LDN   %paruser.buser.1   ** Bloccaggi Doppio
JMPC  NO_LOCK

LD    10000000
DIV   4095
MUL   ANIN2              ** Ingresso analogico Pin 2
DIV   1000
LT    V_MIN_CLOSE_TOOLS  ** Tensione Minima per Attivazione Pompa
S     PUMP_ON_PUNCH_HOLDER ** Uscita Attivazione Pompa Bloccaggi Superiori

LD    10000000
DIV   4095
MUL   ANIN2              ** Ingresso analogico Pin 2
DIV   1000
GT    V_MAX_CLOSE_TOOLS  ** Tensione Massima per Attivazione Pompa
R     PUMP_ON_PUNCH_HOLDER ** Uscita Attivazione Pompa Bloccaggi Superiori

LD    10000000
DIV   4095
MUL   ANIN3              ** Ingresso analogico Pin 3
DIV   1000
LT    V_MIN_CLOSE_TOOLS  ** Tensione Minima per Attivazione Pompa
S     PUMP_ON_DIE_HOLDER ** Uscita Attivazione Pompa Bloccaggi Inferiori o Bloccaggio Singolo

LD    10000000
DIV   4095
MUL   ANIN3              ** Ingresso analogico Pin 3
DIV   1000
GT    V_MAX_CLOSE_TOOLS  ** Tensione Massima per Attivazione Pompa
R     PUMP_ON_DIE_HOLDER ** Uscita Attivazione Pompa Bloccaggi Inferiori o Bloccaggio Singolo

LD    10000000
DIV   4095
MUL   ANIN2              ** Ingresso analogico Pin 2
DIV   1000
GT    V_TOOLS_OPENED     ** Tensione Utensili Aperti
AND   (
LD    10000000
DIV   4095
MUL   ANIN3              ** Ingresso analogico Pin 3
DIV   1000
GT    V_TOOLS_OPENED     ** Tensione Utensili Aperti
)
ST    HOLDER_OPENED      ** Uscita Bloccaggi Aperti

LD    10000000
DIV   4095
MUL   ANIN2              ** Ingresso analogico Pin 2
DIV   1000
GT    V_TOOLS_OPENED     ** Tensione Utensili Aperti
ST    PUNCH_HOLDER_OPENED ** Uscita Bloccaggi Superiori Aperti

LD    10000000
DIV   4095
MUL   ANIN3              ** Ingresso analogico Pin 3
DIV   1000
GT    V_TOOLS_OPENED     ** Tensione Utensili Aperti
ST    DIE_HOLDER_OPENED  ** Uscita Bloccaggi Inferiori Aperti

NO_LOCK:

*****Fine Gestione Bloccaggi*****

LD    5
ST    %UPLCVERS   * Versione PLC

LD    0
ST    %UPLCREL    * Release PLC

LDN   %IW3.15     	*  Fusibiliera Elettronica
ST    %PLCerr3.15

LDN   %IW3.14	  	*  Sequenza Fasi
ST    %PLCerr3.14

LDN   %IW3.13	 	*  Scatto Termico Bloccaggi
ST    %PLCerr3.13

*LDN   %IW3.12	  	*  Scatto termico Bombatura
*ST    %PLCerr3.12

END_FUNCTION
